(* CoDeSys 2.3 export: STANDARDTYPESALIAS.EXP *)

(* Data type *)
TYPE StandardTypesAlias : ST_StandardTypes; END_TYPE
